FUNCTION_BLOCK SoEResetProcess EXTENDS BaseProcess
VAR_INPUT
	///ADS error ID 
	adsErrorId: UINT;
	///Sercos error ID 
	sercosErrorId: UINT;
END_VAR
VAR_OUTPUT
END_VAR
VAR_IN_OUT
END_VAR
VAR
END_VAR

IF do_request THEN
    do_request_result := request();
    do_request := FALSE;
END_IF;
SUPER^();

{attribute 'TcRpcEnable' := '1'}
METHOD request : RequestResults
VAR_INPUT
END_VAR
VAR_OUTPUT
END_VAR
VAR_IN_OUT
END_VAR
VAR
END_VAR
IF THIS^.statuses.enabledStatus.enabled THEN
    THIS^.start();
    request := RequestResults.ACCEPTED;
ELSE
    request := RequestResults.REJECTED;
END_IF;
END_METHOD

{attribute 'TcRpcEnable' := '1'}
METHOD start
VAR_INPUT
END_VAR
VAR_OUTPUT
END_VAR
VAR_IN_OUT
END_VAR
VAR
END_VAR
THIS^.statuses.busyStatus( isBusy := TRUE );
THIS^.statuses.healthStatus( isGood := TRUE );
END_METHOD

END_FUNCTION_BLOCK

(* stored: Version 1.1.0.1, ProductVersion 3.1.4019.2
   POU SoEResetProcess: Id {bfb7c30f-376d-44ba-abf1-ae9696664086}, SpecialFunc None
   Method request: Id {8c98654a-43be-4d96-be6d-af37c5f171de}
   Method start: Id {ed15d89b-8625-4326-9f39-9cb260a0a2be} *)
